// TIA Portal V17 export
// export: Created 2024-01-30T08:49:14.6739582Z, ExportSetting WithDefaults, DisplayName Totally Integrated Automation Portal, DisplayVersion V17 Update 6, DisplayName TIA Portal Openness, DisplayVersion V17 Update 6, DisplayName TIA Portal Version Control Interface, DisplayVersion V17, DisplayName STEP 7 Professional, DisplayVersion V17 Update 6, DisplayName STEP 7 Safety, DisplayVersion V17 Update 6, DisplayName WinCC Advanced, DisplayVersion V17 Update 6
DATA_BLOCK "GDB_Database"   // DB7
{ S7_Optimized_Access := 'TRUE' }
VERSION : 0.1
// stored: AutoNumber true, DBAccessibleFromOPCUA true, DBAccessibleFromWebserver true, IsOnlyStoredInLoadMemory false, IsRetainMemResEnabled false, IsWriteProtectedInAS false, MemoryReserve 100
   VAR
      Communication : Struct   // Communication_Status
         Error : Int;
         Active : Bool;
         Start : Bool;
         Function : Int;
         "Step" : Int;
         Done : Int;
      END_STRUCT;
      Condition : Struct
         Rob_PrgNmr : Int;
      END_STRUCT;
      Receive : Struct
         Rob_PRG : Int;
         Force : Real;
      END_STRUCT;
      Task_Done : Struct
         Read_from_DB : Bool;
      END_STRUCT;
      "Return" : Struct
         t : Bool;
      END_STRUCT;
      Requests : Struct
         Read_from_DB : Bool;
         Write_to_DB : Bool;
      END_STRUCT;
   END_VAR
BEGIN
END_DATA_BLOCK
